FUNCTION_BLOCK FB_LastTimesStats EXTENDS FB_BasicStatistics
VAR_INPUT
	enable: BOOL;	//Enable time counting
END_VAR
VAR_OUTPUT
	lastTime:TIME;
	currTime:TIME;
	lastTimes:ARRAY[1..GVL_Const.lastStatsValue] OF TIME;
	arLastTimes:ARRAY[1..GVL_Const.lastStatsValue] OF LREAL;
END_VAR
VAR
	t1:TON;
	disableTrig:F_TRIG;
	i: UDINT;
END_VAR

disableTrig(CLK:= enable);
IF disableTrig.Q THEN
	lastTime:= t1.ET;
	FOR i:= GVL_Const.lastStatsValue TO 2 BY -1 DO
		lastTimes[i]:= lastTimes[i-1];
	END_FOR
	lastTimes[1]:=lastTime;
	FOR i:= 1 TO GVL_Const.lastStatsValue DO
		arLastTimes[i]:= TIME_TO_LREAL(lastTimes[i])/1000;
	END_FOR
END_IF
t1(IN:= enable, PT:= T#7D);
currTime:= t1.ET;

METHOD M_GetBasicStats : ST_BasicStats
VAR_INPUT
END_VAR
M_GetBasicStats.avg:=SUPER^.M_CalcAvg(THIS^.arLastTimes);
M_GetBasicStats.maximum:=SUPER^.M_CalcMax(THIS^.arLastTimes);
M_GetBasicStats.minimum:=SUPER^.M_CalcMin(THIS^.arLastTimes);
M_GetBasicStats.variance:=SUPER^.M_CalcVariance(THIS^.arLastTimes);
M_GetBasicStats.standardDeviation:=SUPER^.M_CalcSD(THIS^.arLastTimes);
END_METHOD

END_FUNCTION_BLOCK

(* stored: Version 1.1.0.1, ProductVersion 3.1.4024.11
   POU FB_LastTimesStats: Id {114b52f8-2a30-491f-b01f-6fcf6d354093}, SpecialFunc None
   Method M_GetBasicStats: Id {4423bfc3-d543-436b-b7ff-b92f25c2aa18} *)
